// TIA Portal V20 export
DATA_BLOCK "SP201"   // DB312
// stored: MemoryReserve 100
   VAR
      "MAIN OP AUTO INITIATE PBL (GREEN)" : Bool;
      "MAIN OP STOP PBL (RED)" : Bool;
      SPARE_12 : Bool;
      SPARE : Bool;
      SPARE_1 : Bool;
      SPARE_2 : Bool;
      SPARE_3 : Bool;
      SPARE_4 : Bool;
      "MAIN HMI POWER TRIPPED E110CB" : Bool;
      SPARE_5 : Bool;
      SPARE_6 : Bool;
      SPARE_7 : Bool;
      SPARE_8 : Bool;
      SPARE_9 : Bool;
      SPARE_10 : Bool;
      SPARE_11 : Bool;
   END_VAR
BEGIN
END_DATA_BLOCK
